Fanuc KAREL source: kt00166.KL

-- PROVISIONAL review KL for V770-1; original PC SHA256 f719b89f0d845596735199d6162ef9e70230ff341e80dbe467ab90a37f1b6229
-- Incomplete behavior may be omitted. Consult companion uncertainty JSON. Do not deploy.
PROGRAM KT00166
%NOLOCKGROUP
VAR
  I1 : INTEGER
  OUT : REAL
-- UNRESOLVED_DECL Y2 type=002018
BEGIN
  -- UNRESOLVED_PC offsets 5-16; opcodes 2E,23
  -- UNRESOLVED_PC offsets 21-35; opcodes 2E,22,9D,33,B2
  -- UNRESOLVED_PC offsets 40-63; opcodes 21,22,9D,33,B1,56,64,23
  -- UNRESOLVED_PC offsets 68-72; opcodes 7F
END KT00166
